FUNCTION_BLOCK LfcPrint
  (* Standard: 61499-2 *)
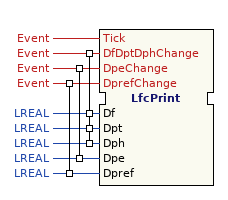
  EVENT_INPUT
    Tick;
    DfDptDphChange WITH Df, Dpt, Dph;
    DpeChange WITH Dpe;
    DprefChange WITH Dpref;
  END_EVENT
  VAR_INPUT
    Df : LREAL;
    Dpt : LREAL;
    Dph : LREAL;
    Dpe : LREAL;
    Dpref : LREAL;
  END_VAR
END_FUNCTION_BLOCK
(* other elements stored in the file *)
(* Autogenerate Language=C ArbitraryText= #include <stdio.h> #include <stdlib.h> RunText= static int tickCount = 0; printf("%10f, %10f Hz, %10f MW Generation, %10f MW Load, %10f, %10f, %10f, %10f\r\n", tickCount * 0.0001, me->Df + 60, 1000 + me->Dpt * 1000, 1000 + me->Dpe * 1000, me->Dpref, me->Df, me->Dpt, me->Dph); tickCount++; *)
